Omron CX-Programmer project NewProject (CX-Programmer 9.75)

# PLC NewPLC1: CP1H XA

## Global symbols (name address type ; comment)
0 CHANNEL  ; ASSEMBLED AND DISSASSEMBLED
13.01 BOOL  ; FRGTGHN
13.05 BOOL  ; reset1
17.02 BOOL  ; reset2
265.00 BOOL  ; FEEDING BASE HMI
266.00 BOOL  ; ASSEMBLING THE BEARING
267.01 BOOL  ; INSERTION OF THE SHAFT
269.00 BOOL  ; POSITIONING OF THE COVER
278.00 BOOL  ; RUN
400.00 BOOL  ; run
C0000 BOOL  ; cup
D100 CHANNEL  ; MOV2
D105 CHANNEL  ; MOV1
D80 CHANNEL  ; .....
T0030 BOOL  ; TIMER30
W0 CHANNEL  ; ..;;,
W1 CHANNEL  ; EF

## Program NewProgram1 (cyclic task 0)
Local symbols
APLUS 100.00 BOOL  ; Feeder cylinder forwards
BPLUS 100.01 BOOL  ; Body transfer cylinder forwards
CPLUS 100.02 BOOL  ; Position verification cylinder downwards
DPLUS 100.03 BOOL  ; Rejection cylinder forwards
EMINUS 100.05 BOOL  ; Rotary actuator backwards
EPLUS 100.04 BOOL  ; Rotary actuator forwards
FM 101.06 BOOL  ; Error light on
FPLUS 100.06 BOOL  ; Opening of the gripper of the rotary actuator
GPLUS 100.07 BOOL  ; Shaft insertion manipulator downwards
HPLUS 101.00 BOOL  ; Shaft insertion manipulator forwards
IPLUS 101.01 BOOL  ; Gripper closure
JMINUS 101.03 BOOL  ; Cover insertion manipulator backwards
JPLUS 101.02 BOOL  ; Cover insertion manipulator forwards
KPLUS 101.04 BOOL  ; Cover insertion manipulator downwards
Step_0 H0.00 BOOL  ; Step 0
Step_1 H0.01 BOOL  ; Step  1
Step_10 H0.10 BOOL  ; Step 10
Step_11 H0.11 BOOL  ; Step 11
Step_12 H0.12 BOOL  ; Step 12
Step_13 H0.13 BOOL  ; Step 13
Step_14 H0.14 BOOL  ; Step 14
Step_15 H0.15 BOOL  ; Step 15
Step_16 H1.00 BOOL  ; Step 16
Step_17 H1.01 BOOL  ; Step 17
Step_18 H1.02 BOOL  ; Step 18
Step_19 H1.03 BOOL  ; Step 19
Step_2 H0.02 BOOL  ; Step 2
Step_20 H1.04 BOOL  ; Step 20
Step_21 H1.05 BOOL  ; Step 21
Step_22 H1.06 BOOL  ; Step 22
Step_23 H1.07 BOOL  ; Step 23
Step_24 H1.08 BOOL  ; Step 24
Step_25 H1.09 BOOL  ; Step 25
Step_26 H1.10 BOOL  ; Step 26
Step_27 H1.11 BOOL  ; Step 27
Step_28 H1.12 BOOL  ; Step 28
Step_29 H1.13 BOOL  ; Step 29
Step_3 H0.03 BOOL  ; Step 3
Step_30 H1.14 BOOL  ; Step 30
Step_31 H1.15 BOOL  ; Step 31
Step_32 H2.00 BOOL  ; Step 32
Step_33 H2.01 BOOL  ; Step 33
Step_34 H2.02 BOOL  ; Step 34
Step_35 H2.03 BOOL  ; Step 35
Step_36 H2.04 BOOL  ; Step 36
Step_37 H2.05 BOOL  ; Step 37
Step_38 H2.06 BOOL  ; Step 38
Step_39 H2.07 BOOL  ; Step 39
Step_4 H0.04 BOOL  ; Step 4
Step_40 H2.08 BOOL  ; Step 40
Step_41 H2.09 BOOL  ; Step 41
Step_42 H2.10 BOOL  ; Step 42
Step_43 H2.11 BOOL  ; Step 43
Step_44 H2.12 BOOL  ; Step 44
Step_45 H2.13 BOOL  ; Step 45
Step_46 H2.14 BOOL  ; Step 46
Step_47 H2.15 BOOL  ; Step 47
Step_48 H3.00 BOOL  ; Step 48
Step_49 H3.01 BOOL  ; Step 49
Step_5 H0.05 BOOL  ; Step 5
Step_50 H3.02 BOOL  ; Step 50
Step_51 H3.03 BOOL  ; Step 51
Step_6 H0.06 BOOL  ; Step 6
Step_60 H3.04 BOOL  ; Step 60
Step_61 H3.05 BOOL  ; Step 61
Step_62 H3.06 BOOL  ; Step 62
Step_7 H0.07 BOOL  ; Step 7
Step_8 H0.08 BOOL  ; Step 8
Step_9 H0.09 BOOL  ; Step 9
VPLUS 101.05 BOOL  ; Vacuum in cups
a_0 0.03 BOOL  ; Body Feeder backward
a_1 0.04 BOOL  ; Body Feeder forward
am_SCADA 20.02 BOOL  ; Auto/manu selector from SCADA
atm 0.02 BOOL  ; Auto/Manu selector
b_1 0.05 BOOL  ; Body transfer cylinder forward
bearing_placed 200.10 BOOL  ; bearing placed on body
body_ok 200.04 BOOL  ; Body placed ok
c_1 0.06 BOOL  ; Position verification cylinder downward
continue 200.01 BOOL  ; Continue cycle from one step to another
cover 200.02 BOOL  ; cover in position
cover_placed 200.09 BOOL  ; cover placed on body
cycle H4.00 BOOL  ; Cycle started
cycle_end 200.11 BOOL  ; cycle end
cycle_start 30.07 BOOL  ; cycle start
dp1 1.09 BOOL  ; Body detector
dp2 1.10 BOOL  ; Bearing detector
dp3 1.11 BOOL  ; Shaft detector
dp4 200.08 BOOL  ; Cover detector
e_0 0.07 BOOL  ; Rotary actuator backward
e_1 0.08 BOOL  ; Rotary actuator in the middle position
e_2 0.09 BOOL  ; Rotary actuator forward
error 200.12 BOOL  ; Error in the station
g_0 0.10 BOOL  ; Shaft insertion manipulator upward
g_1 0.11 BOOL  ; Shaft insertion manipulator downward
h_0 1.00 BOOL  ; Shaft insertion manipulator backward
h_1 1.01 BOOL  ; Shaft insertion manipulator forward
i_0 1.02 BOOL  ; Gripper opened
i_1 1.03 BOOL  ; Gripper closed
i_c 200.03 BOOL  ; Initial condition
j_0 1.04 BOOL  ; Cover insertion manipulator backward
j_1 1.05 BOOL  ; Cover insertion manipulator forward
k_0 1.06 BOOL  ; Cover insertion manipulator upward
k_1 1.07 BOOL  ; Cover insertion manipulator downward
m 0.00 BOOL  ; Start button
m_SCADA 20.00 BOOL  ; Start button fron Scada
no_air_pressure 200.06 BOOL  ; No air pressure
no_e1 200.07 BOOL  ; Initial condition of bearing manipulator
on 200.00 BOOL  ; Start in auto mode
p 0.01 BOOL  ; Stop button
p_SCADA 20.01 BOOL  ; Stop button from Scada
shaft_placed 200.13 BOOL  ; shaft placed on body
t_0_PV T0 CHANNEL  ; Timer 0
t_0_step T0000 BOOL  ; Timer 0
t_10_PV T10 CHANNEL  ; Timer 10
t_10_step T0010 BOOL  ; Timer 10
t_11_step T0011 BOOL  ; Timer 11
t_12_step T0012 BOOL  ; Timer 12
t_13_step T0013 BOOL  ; Timer 13
t_14_step T0014 BOOL  ; Timer 14
t_15 T0015 BOOL  ; Timer 15
t_16 T0016 BOOL  ; Timer 16
t_17 T0017 BOOL  ; Timer 17
t_18 T0018 BOOL  ; Timer 18
t_19 T0019 BOOL  ; Timer 19
t_1_PV T1 CHANNEL  ; Timer 1
t_1_step T0001 BOOL  ; Timer 1
t_20 T0020 BOOL  ; Timer 20
t_21 T0021 BOOL  ; Timer 21
t_22 T0022 BOOL  ; Timer 22
t_23 T0023 BOOL  ; Timer 23
t_24 T0024 BOOL  ; Timer 24
t_2_PV T2 CHANNEL  ; Timer 2
t_2_step T0002 BOOL  ; Timer 2
t_3_PV T3 CHANNEL  ; Timer 3
t_3_step T0003 BOOL  ; Timer 3
t_4_PV T4 CHANNEL  ; Timer 4
t_4_step T0004 BOOL  ; Timer 4
t_5_PV T5 CHANNEL  ; Timer 5
t_5_step T0005 BOOL  ; Timer 5
t_6_PV T6 CHANNEL  ; Timer 6
t_6_step T0006 BOOL  ; Timer 6
t_7 BOOL
t_7_PV T7 CHANNEL  ; Timer 7
t_7_step T0007 BOOL  ; Timer 7
t_8_PV T8 CHANNEL  ; Timer 8
t_8_step T0008 BOOL  ; Timer 8
t_9_PV T9 CHANNEL  ; Timer 9
t_9_step T0009 BOOL  ; Timer 9
v 1.08 BOOL  ; Vacuum in cups
wait 200.05 BOOL  ; Wait to return subroutine

### Section Steps

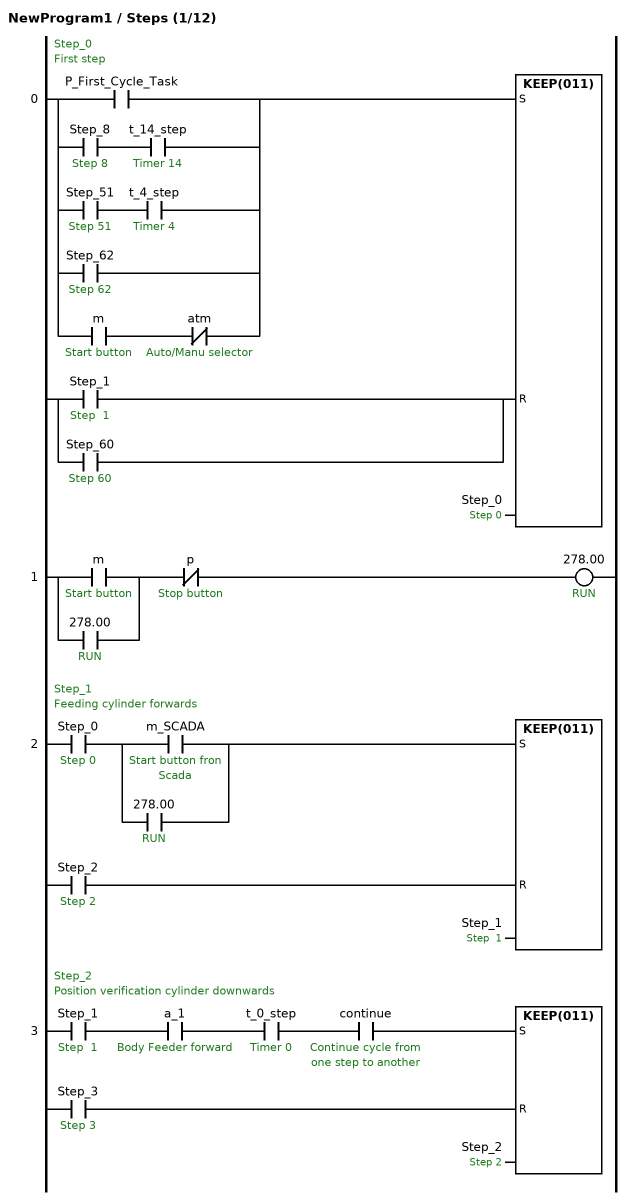
; rung 0: Step_0 / First step
LD P_First_Cycle_Task
LD Step_8  ; Step 8
AND t_14_step  ; Timer 14
ORLD
LD Step_51  ; Step 51
AND t_4_step  ; Timer 4
ORLD
OR Step_62  ; Step 62
LD m  ; Start button
ANDNOT atm  ; Auto/Manu selector
ORLD
LD Step_1  ; Step  1
OR Step_60  ; Step 60
KEEP(011) Step_0  ; Step 0
; rung 1
LD m  ; Start button
OR 278.00  ; RUN
ANDNOT p  ; Stop button
OUT 278.00  ; RUN
; rung 2: Step_1 / Feeding cylinder forwards
LD Step_0  ; Step 0
LD m_SCADA  ; Start button fron Scada
OR 278.00  ; RUN
ANDLD
LD Step_2  ; Step 2
KEEP(011) Step_1  ; Step  1
; rung 3: Step_2 / Position verification cylinder downwards
LD Step_1  ; Step  1
AND a_1  ; Body Feeder forward
AND t_0_step  ; Timer 0
AND continue  ; Continue cycle from one step to another
LD Step_3  ; Step 3
KEEP(011) Step_2  ; Step 2

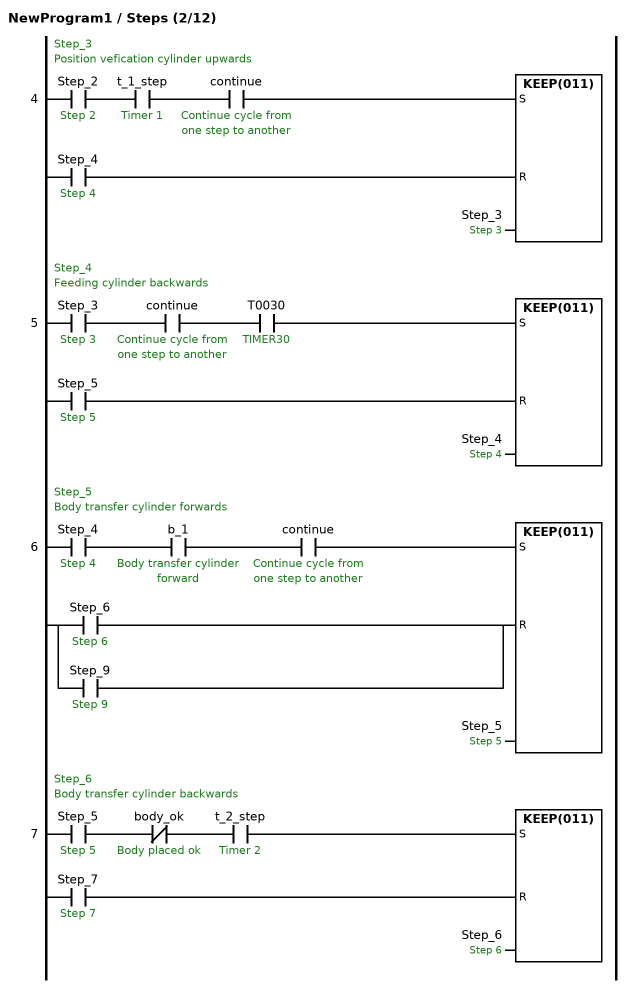
; rung 4: Step_3 / Position vefication cylinder upwards
LD Step_2  ; Step 2
AND t_1_step  ; Timer 1
AND continue  ; Continue cycle from one step to another
LD Step_4  ; Step 4
KEEP(011) Step_3  ; Step 3
; rung 5: Step_4 / Feeding cylinder backwards
LD Step_3  ; Step 3
AND continue  ; Continue cycle from one step to another
AND T0030  ; TIMER30
LD Step_5  ; Step 5
KEEP(011) Step_4  ; Step 4
; rung 6: Step_5 / Body transfer cylinder forwards
LD Step_4  ; Step 4
AND b_1  ; Body transfer cylinder forward
AND continue  ; Continue cycle from one step to another
LD Step_6  ; Step 6
OR Step_9  ; Step 9
KEEP(011) Step_5  ; Step 5
; rung 7: Step_6 / Body transfer cylinder backwards
LD Step_5  ; Step 5
ANDNOT body_ok  ; Body placed ok
AND t_2_step  ; Timer 2
LD Step_7  ; Step 7
KEEP(011) Step_6  ; Step 6

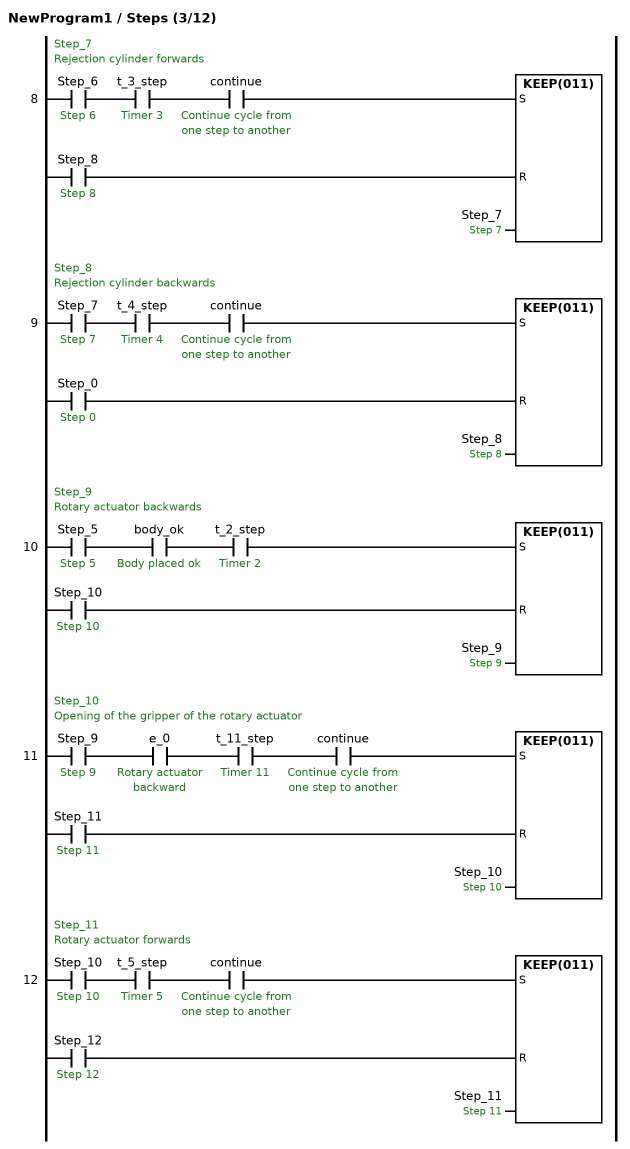
; rung 8: Step_7 / Rejection cylinder forwards
LD Step_6  ; Step 6
AND t_3_step  ; Timer 3
AND continue  ; Continue cycle from one step to another
LD Step_8  ; Step 8
KEEP(011) Step_7  ; Step 7
; rung 9: Step_8 / Rejection cylinder backwards
LD Step_7  ; Step 7
AND t_4_step  ; Timer 4
AND continue  ; Continue cycle from one step to another
LD Step_0  ; Step 0
KEEP(011) Step_8  ; Step 8
; rung 10: Step_9 / Rotary actuator backwards
LD Step_5  ; Step 5
AND body_ok  ; Body placed ok
AND t_2_step  ; Timer 2
LD Step_10  ; Step 10
KEEP(011) Step_9  ; Step 9
; rung 11: Step_10 / Opening of the gripper of the rotary actuator
LD Step_9  ; Step 9
AND e_0  ; Rotary actuator backward
AND t_11_step  ; Timer 11
AND continue  ; Continue cycle from one step to another
LD Step_11  ; Step 11
KEEP(011) Step_10  ; Step 10
; rung 12: Step_11 / Rotary actuator forwards
LD Step_10  ; Step 10
AND t_5_step  ; Timer 5
AND continue  ; Continue cycle from one step to another
LD Step_12  ; Step 12
KEEP(011) Step_11  ; Step 11

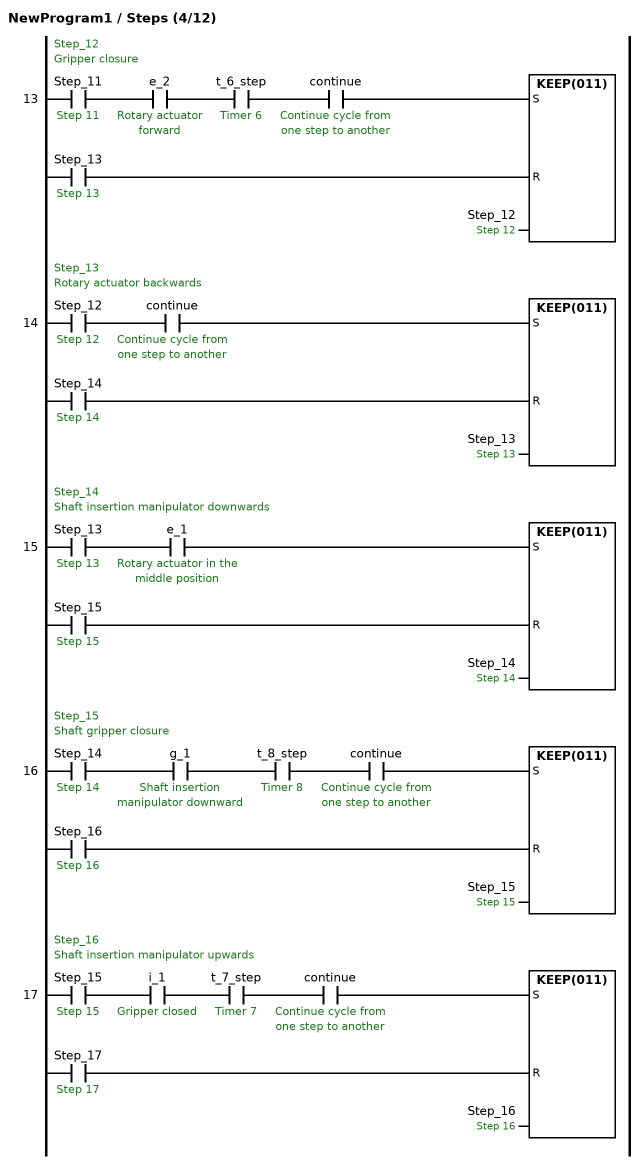
; rung 13: Step_12 / Gripper closure
LD Step_11  ; Step 11
AND e_2  ; Rotary actuator forward
AND t_6_step  ; Timer 6
AND continue  ; Continue cycle from one step to another
LD Step_13  ; Step 13
KEEP(011) Step_12  ; Step 12
; rung 14: Step_13 / Rotary actuator backwards
LD Step_12  ; Step 12
AND continue  ; Continue cycle from one step to another
LD Step_14  ; Step 14
KEEP(011) Step_13  ; Step 13
; rung 15: Step_14 / Shaft insertion manipulator downwards
LD Step_13  ; Step 13
AND e_1  ; Rotary actuator in the middle position
LD Step_15  ; Step 15
KEEP(011) Step_14  ; Step 14
; rung 16: Step_15 / Shaft gripper closure
LD Step_14  ; Step 14
AND g_1  ; Shaft insertion manipulator downward
AND t_8_step  ; Timer 8
AND continue  ; Continue cycle from one step to another
LD Step_16  ; Step 16
KEEP(011) Step_15  ; Step 15
; rung 17: Step_16 / Shaft insertion manipulator upwards
LD Step_15  ; Step 15
AND i_1  ; Gripper closed
AND t_7_step  ; Timer 7
AND continue  ; Continue cycle from one step to another
LD Step_17  ; Step 17
KEEP(011) Step_16  ; Step 16

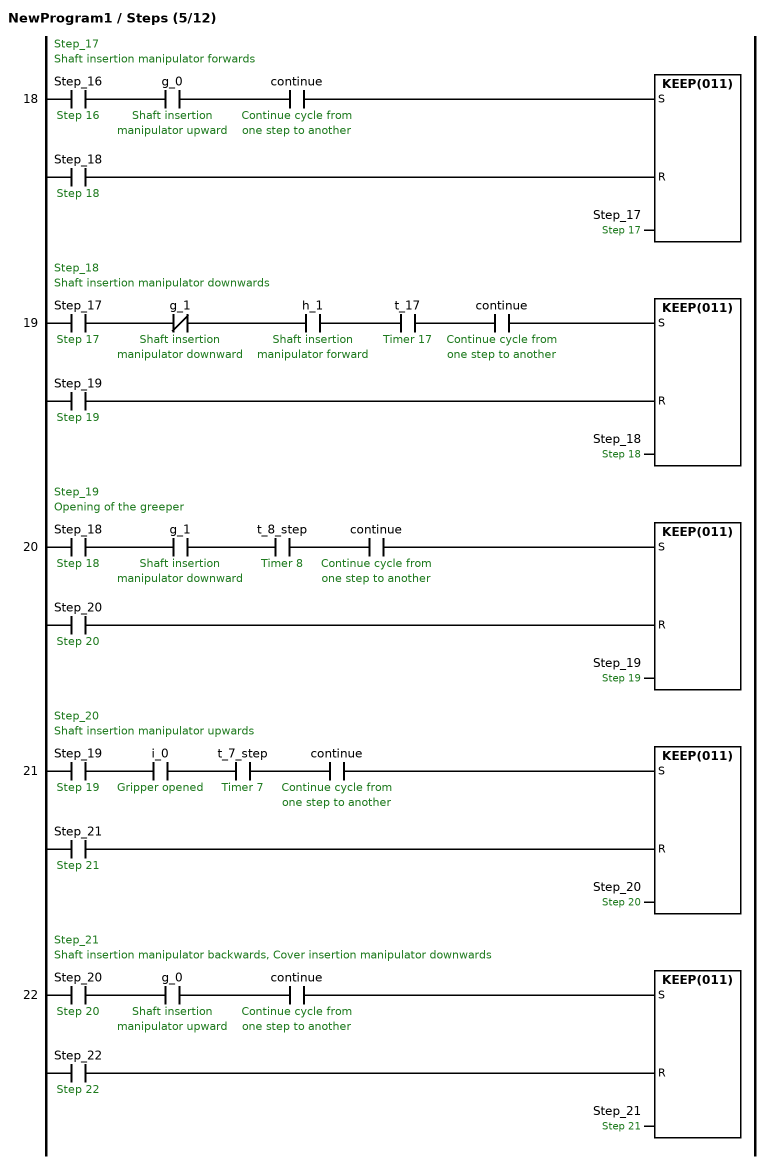
; rung 18: Step_17 / Shaft insertion manipulator forwards
LD Step_16  ; Step 16
AND g_0  ; Shaft insertion manipulator upward
AND continue  ; Continue cycle from one step to another
LD Step_18  ; Step 18
KEEP(011) Step_17  ; Step 17
; rung 19: Step_18 / Shaft insertion manipulator downwards
LD Step_17  ; Step 17
ANDNOT g_1  ; Shaft insertion manipulator downward
AND h_1  ; Shaft insertion manipulator forward
AND t_17  ; Timer 17
AND continue  ; Continue cycle from one step to another
LD Step_19  ; Step 19
KEEP(011) Step_18  ; Step 18
; rung 20: Step_19 / Opening of the greeper
LD Step_18  ; Step 18
AND g_1  ; Shaft insertion manipulator downward
AND t_8_step  ; Timer 8
AND continue  ; Continue cycle from one step to another
LD Step_20  ; Step 20
KEEP(011) Step_19  ; Step 19
; rung 21: Step_20 / Shaft insertion manipulator upwards
LD Step_19  ; Step 19
AND i_0  ; Gripper opened
AND t_7_step  ; Timer 7
AND continue  ; Continue cycle from one step to another
LD Step_21  ; Step 21
KEEP(011) Step_20  ; Step 20
; rung 22: Step_21 / Shaft insertion manipulator backwards, Cover insertion manipulator downwards
LD Step_20  ; Step 20
AND g_0  ; Shaft insertion manipulator upward
AND continue  ; Continue cycle from one step to another
LD Step_22  ; Step 22
KEEP(011) Step_21  ; Step 21

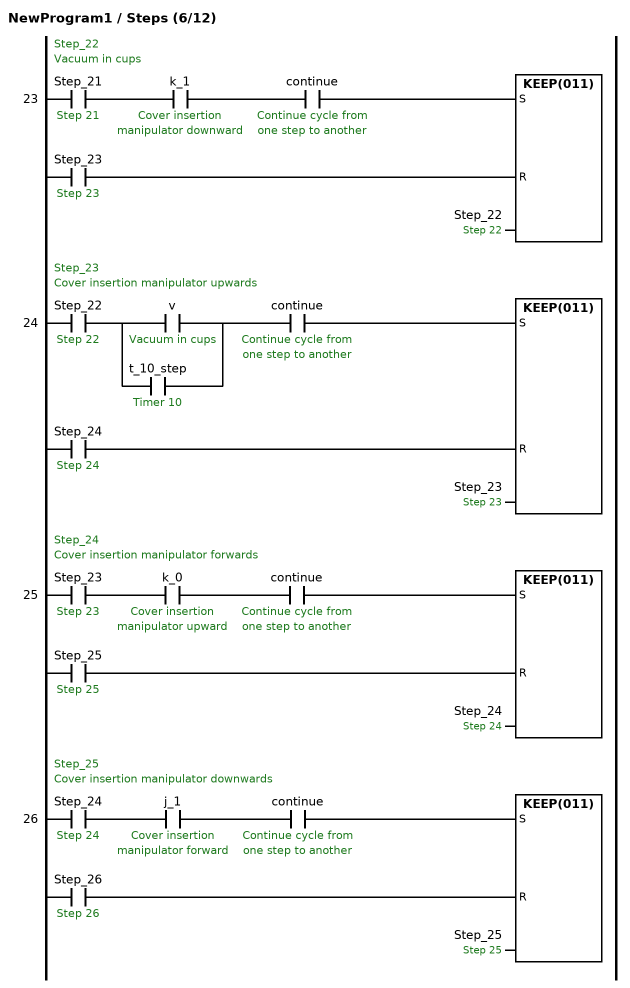
; rung 23: Step_22 / Vacuum in cups
LD Step_21  ; Step 21
AND k_1  ; Cover insertion manipulator downward
AND continue  ; Continue cycle from one step to another
LD Step_23  ; Step 23
KEEP(011) Step_22  ; Step 22
; rung 24: Step_23 / Cover insertion manipulator upwards
LD Step_22  ; Step 22
LD v  ; Vacuum in cups
OR t_10_step  ; Timer 10
ANDLD
AND continue  ; Continue cycle from one step to another
LD Step_24  ; Step 24
KEEP(011) Step_23  ; Step 23
; rung 25: Step_24 / Cover insertion manipulator forwards
LD Step_23  ; Step 23
AND k_0  ; Cover insertion manipulator upward
AND continue  ; Continue cycle from one step to another
LD Step_25  ; Step 25
KEEP(011) Step_24  ; Step 24
; rung 26: Step_25 / Cover insertion manipulator downwards
LD Step_24  ; Step 24
AND j_1  ; Cover insertion manipulator forward
AND continue  ; Continue cycle from one step to another
LD Step_26  ; Step 26
KEEP(011) Step_25  ; Step 25

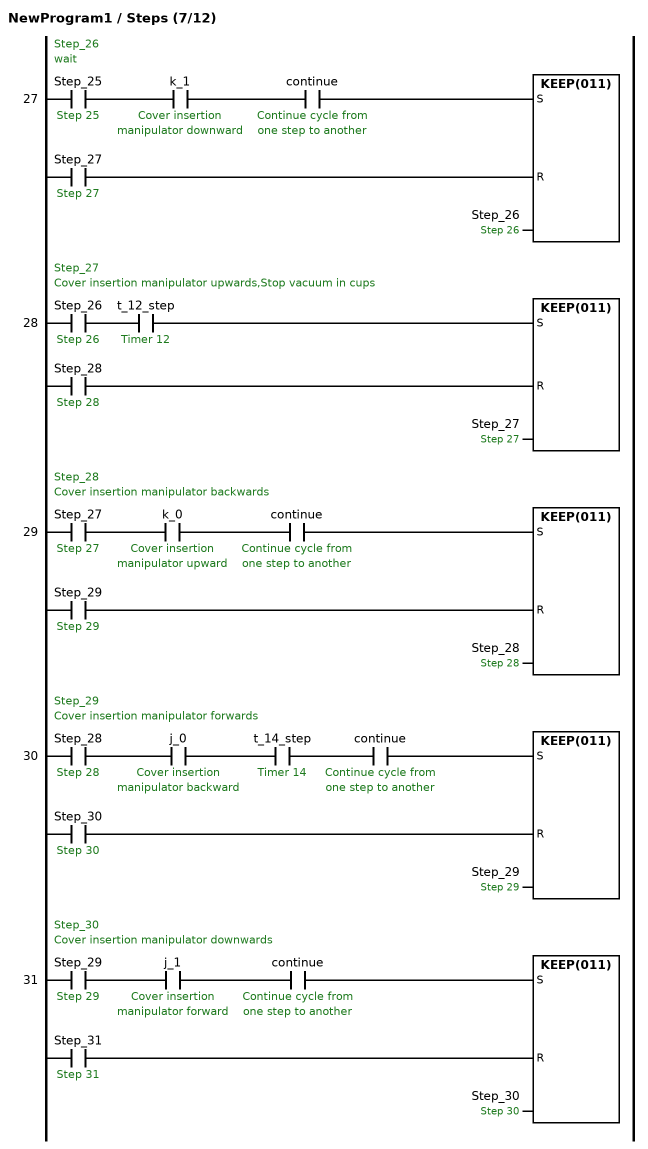
; rung 27: Step_26 / wait
LD Step_25  ; Step 25
AND k_1  ; Cover insertion manipulator downward
AND continue  ; Continue cycle from one step to another
LD Step_27  ; Step 27
KEEP(011) Step_26  ; Step 26
; rung 28: Step_27 / Cover insertion manipulator upwards,Stop vacuum in cups
LD Step_26  ; Step 26
AND t_12_step  ; Timer 12
LD Step_28  ; Step 28
KEEP(011) Step_27  ; Step 27
; rung 29: Step_28 / Cover insertion manipulator backwards
LD Step_27  ; Step 27
AND k_0  ; Cover insertion manipulator upward
AND continue  ; Continue cycle from one step to another
LD Step_29  ; Step 29
KEEP(011) Step_28  ; Step 28
; rung 30: Step_29 / Cover insertion manipulator forwards
LD Step_28  ; Step 28
AND j_0  ; Cover insertion manipulator backward
AND t_14_step  ; Timer 14
AND continue  ; Continue cycle from one step to another
LD Step_30  ; Step 30
KEEP(011) Step_29  ; Step 29
; rung 31: Step_30 / Cover insertion manipulator downwards
LD Step_29  ; Step 29
AND j_1  ; Cover insertion manipulator forward
AND continue  ; Continue cycle from one step to another
LD Step_31  ; Step 31
KEEP(011) Step_30  ; Step 30

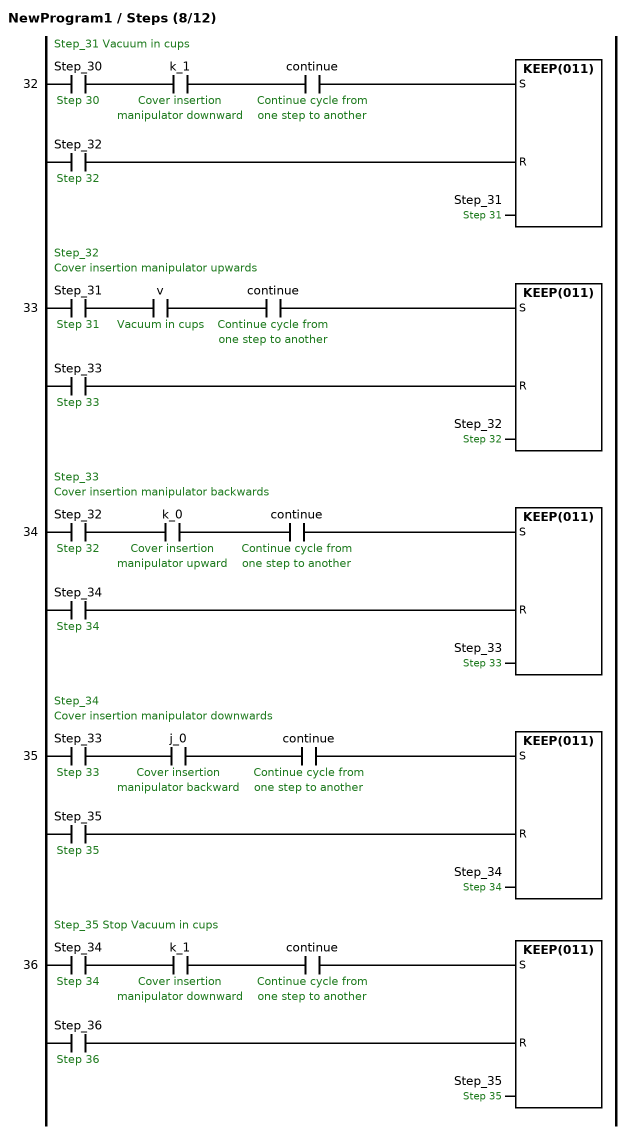
; rung 32: Step_31 Vacuum in cups
LD Step_30  ; Step 30
AND k_1  ; Cover insertion manipulator downward
AND continue  ; Continue cycle from one step to another
LD Step_32  ; Step 32
KEEP(011) Step_31  ; Step 31
; rung 33: Step_32 / Cover insertion manipulator upwards
LD Step_31  ; Step 31
AND v  ; Vacuum in cups
AND continue  ; Continue cycle from one step to another
LD Step_33  ; Step 33
KEEP(011) Step_32  ; Step 32
; rung 34: Step_33 / Cover insertion manipulator backwards
LD Step_32  ; Step 32
AND k_0  ; Cover insertion manipulator upward
AND continue  ; Continue cycle from one step to another
LD Step_34  ; Step 34
KEEP(011) Step_33  ; Step 33
; rung 35: Step_34 / Cover insertion manipulator downwards
LD Step_33  ; Step 33
AND j_0  ; Cover insertion manipulator backward
AND continue  ; Continue cycle from one step to another
LD Step_35  ; Step 35
KEEP(011) Step_34  ; Step 34
; rung 36: Step_35 Stop Vacuum in cups
LD Step_34  ; Step 34
AND k_1  ; Cover insertion manipulator downward
AND continue  ; Continue cycle from one step to another
LD Step_36  ; Step 36
KEEP(011) Step_35  ; Step 35

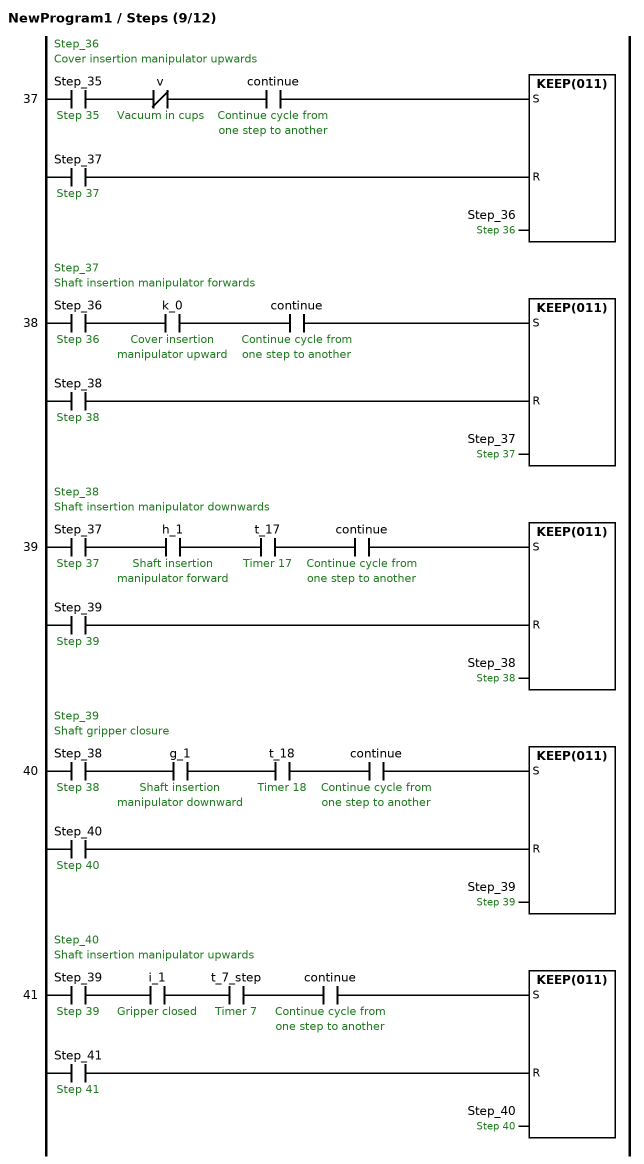
; rung 37: Step_36 / Cover insertion manipulator upwards
LD Step_35  ; Step 35
ANDNOT v  ; Vacuum in cups
AND continue  ; Continue cycle from one step to another
LD Step_37  ; Step 37
KEEP(011) Step_36  ; Step 36
; rung 38: Step_37 / Shaft insertion manipulator forwards
LD Step_36  ; Step 36
AND k_0  ; Cover insertion manipulator upward
AND continue  ; Continue cycle from one step to another
LD Step_38  ; Step 38
KEEP(011) Step_37  ; Step 37
; rung 39: Step_38 / Shaft insertion manipulator downwards
LD Step_37  ; Step 37
AND h_1  ; Shaft insertion manipulator forward
AND t_17  ; Timer 17
AND continue  ; Continue cycle from one step to another
LD Step_39  ; Step 39
KEEP(011) Step_38  ; Step 38
; rung 40: Step_39 / Shaft gripper closure
LD Step_38  ; Step 38
AND g_1  ; Shaft insertion manipulator downward
AND t_18  ; Timer 18
AND continue  ; Continue cycle from one step to another
LD Step_40  ; Step 40
KEEP(011) Step_39  ; Step 39
; rung 41: Step_40 / Shaft insertion manipulator upwards
LD Step_39  ; Step 39
AND i_1  ; Gripper closed
AND t_7_step  ; Timer 7
AND continue  ; Continue cycle from one step to another
LD Step_41  ; Step 41
KEEP(011) Step_40  ; Step 40

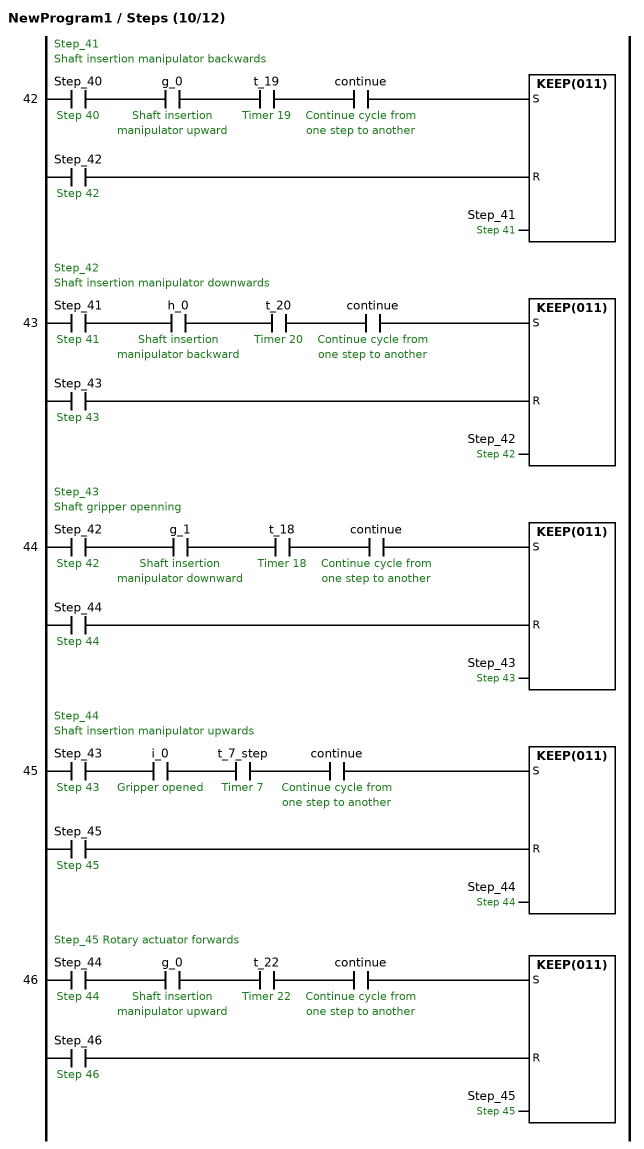
; rung 42: Step_41 / Shaft insertion manipulator backwards
LD Step_40  ; Step 40
AND g_0  ; Shaft insertion manipulator upward
AND t_19  ; Timer 19
AND continue  ; Continue cycle from one step to another
LD Step_42  ; Step 42
KEEP(011) Step_41  ; Step 41
; rung 43: Step_42 / Shaft insertion manipulator downwards
LD Step_41  ; Step 41
AND h_0  ; Shaft insertion manipulator backward
AND t_20  ; Timer 20
AND continue  ; Continue cycle from one step to another
LD Step_43  ; Step 43
KEEP(011) Step_42  ; Step 42
; rung 44: Step_43 / Shaft gripper openning
LD Step_42  ; Step 42
AND g_1  ; Shaft insertion manipulator downward
AND t_18  ; Timer 18
AND continue  ; Continue cycle from one step to another
LD Step_44  ; Step 44
KEEP(011) Step_43  ; Step 43
; rung 45: Step_44 / Shaft insertion manipulator upwards
LD Step_43  ; Step 43
AND i_0  ; Gripper opened
AND t_7_step  ; Timer 7
AND continue  ; Continue cycle from one step to another
LD Step_45  ; Step 45
KEEP(011) Step_44  ; Step 44
; rung 46: Step_45 Rotary actuator forwards
LD Step_44  ; Step 44
AND g_0  ; Shaft insertion manipulator upward
AND t_22  ; Timer 22
AND continue  ; Continue cycle from one step to another
LD Step_46  ; Step 46
KEEP(011) Step_45  ; Step 45

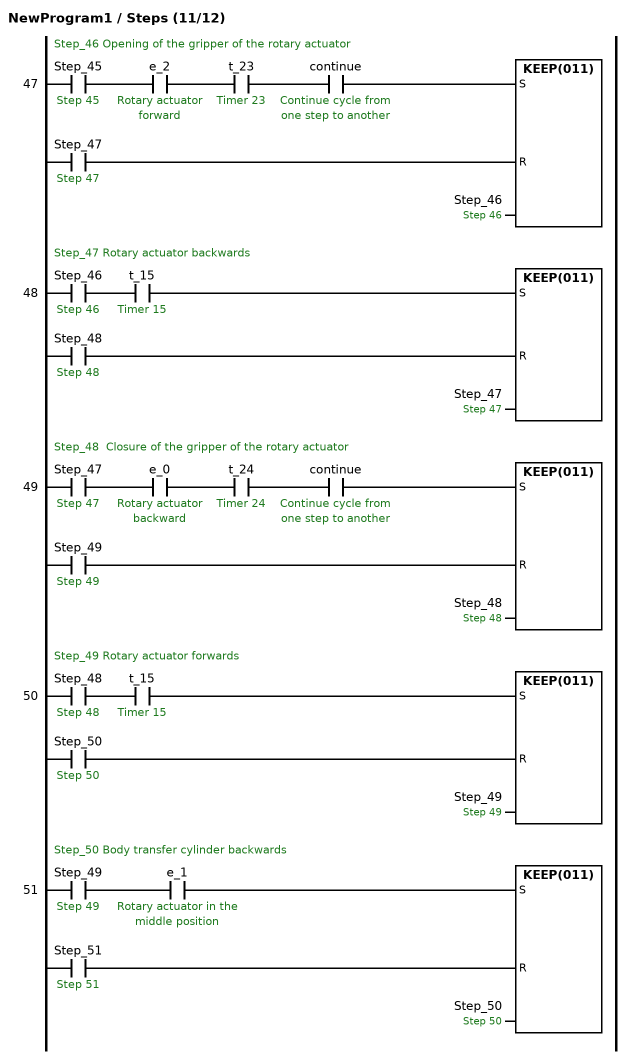
; rung 47: Step_46 Opening of the gripper of the rotary actuator
LD Step_45  ; Step 45
AND e_2  ; Rotary actuator forward
AND t_23  ; Timer 23
AND continue  ; Continue cycle from one step to another
LD Step_47  ; Step 47
KEEP(011) Step_46  ; Step 46
; rung 48: Step_47 Rotary actuator backwards
LD Step_46  ; Step 46
AND t_15  ; Timer 15
LD Step_48  ; Step 48
KEEP(011) Step_47  ; Step 47
; rung 49: Step_48  Closure of the gripper of the rotary actuator
LD Step_47  ; Step 47
AND e_0  ; Rotary actuator backward
AND t_24  ; Timer 24
AND continue  ; Continue cycle from one step to another
LD Step_49  ; Step 49
KEEP(011) Step_48  ; Step 48
; rung 50: Step_49 Rotary actuator forwards
LD Step_48  ; Step 48
AND t_15  ; Timer 15
LD Step_50  ; Step 50
KEEP(011) Step_49  ; Step 49
; rung 51: Step_50 Body transfer cylinder backwards
LD Step_49  ; Step 49
AND e_1  ; Rotary actuator in the middle position
LD Step_51  ; Step 51
KEEP(011) Step_50  ; Step 50

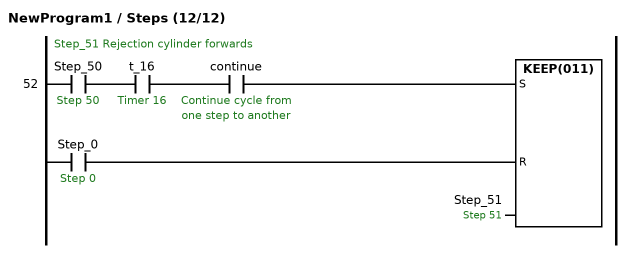
; rung 52: Step_51 Rejection cylinder forwards
LD Step_50  ; Step 50
AND t_16  ; Timer 16
AND continue  ; Continue cycle from one step to another
LD Step_0  ; Step 0
KEEP(011) Step_51  ; Step 51

### Section Outputs

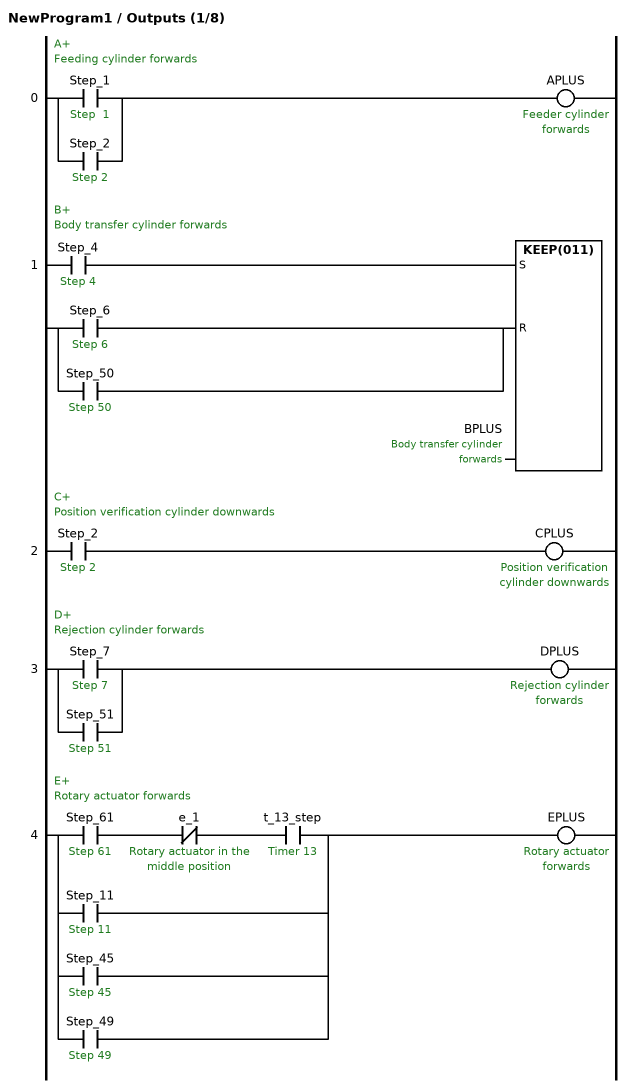
; rung 0: A+ / Feeding cylinder forwards
LD Step_1  ; Step  1
OR Step_2  ; Step 2
OUT APLUS  ; Feeder cylinder forwards
; rung 1: B+ / Body transfer cylinder forwards
LD Step_4  ; Step 4
LD Step_6  ; Step 6
OR Step_50  ; Step 50
KEEP(011) BPLUS  ; Body transfer cylinder forwards
; rung 2: C+ / Position verification cylinder downwards
LD Step_2  ; Step 2
OUT CPLUS  ; Position verification cylinder downwards
; rung 3: D+ / Rejection cylinder forwards
LD Step_7  ; Step 7
OR Step_51  ; Step 51
OUT DPLUS  ; Rejection cylinder forwards
; rung 4: E+ / Rotary actuator forwards
LD Step_61  ; Step 61
ANDNOT e_1  ; Rotary actuator in the middle position
AND t_13_step  ; Timer 13
OR Step_11  ; Step 11
OR Step_45  ; Step 45
OR Step_49  ; Step 49
OUT EPLUS  ; Rotary actuator forwards

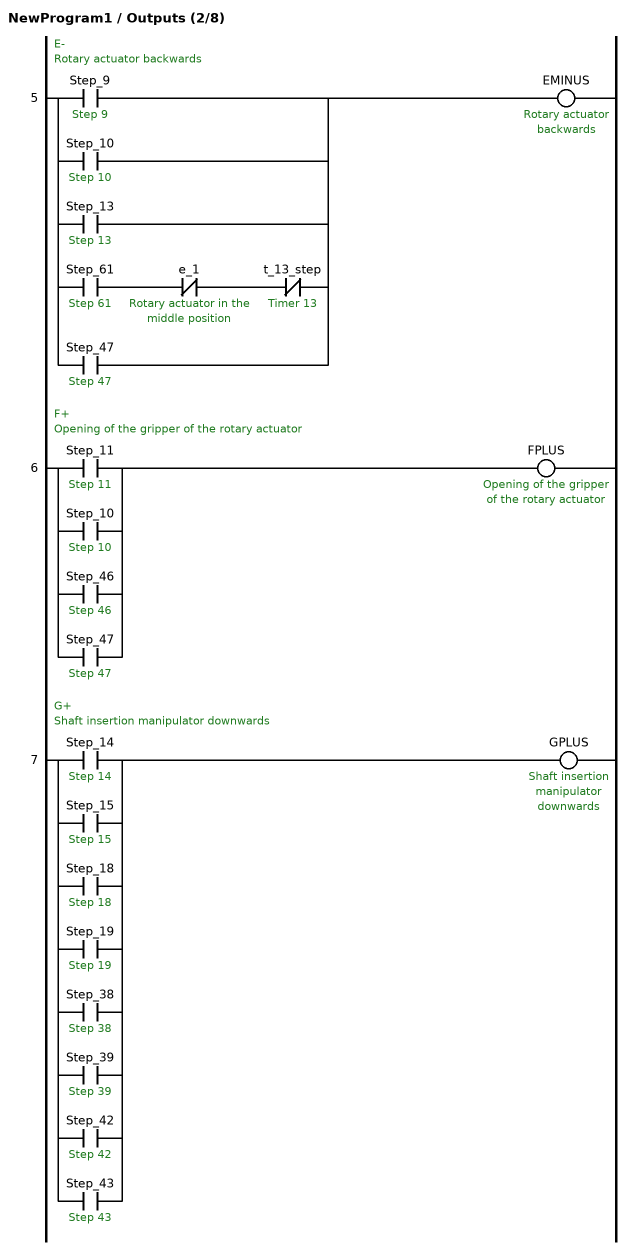
; rung 5: E- / Rotary actuator backwards
LD Step_9  ; Step 9
OR Step_10  ; Step 10
OR Step_13  ; Step 13
LD Step_61  ; Step 61
ANDNOT e_1  ; Rotary actuator in the middle position
ANDNOT t_13_step  ; Timer 13
ORLD
OR Step_47  ; Step 47
OUT EMINUS  ; Rotary actuator backwards
; rung 6: F+ / Opening of the gripper of the rotary actuator
LD Step_11  ; Step 11
OR Step_10  ; Step 10
OR Step_46  ; Step 46
OR Step_47  ; Step 47
OUT FPLUS  ; Opening of the gripper of the rotary actuator
; rung 7: G+ / Shaft insertion manipulator downwards
LD Step_14  ; Step 14
OR Step_15  ; Step 15
OR Step_18  ; Step 18
OR Step_19  ; Step 19
OR Step_38  ; Step 38
OR Step_39  ; Step 39
OR Step_42  ; Step 42
OR Step_43  ; Step 43
OUT GPLUS  ; Shaft insertion manipulator downwards

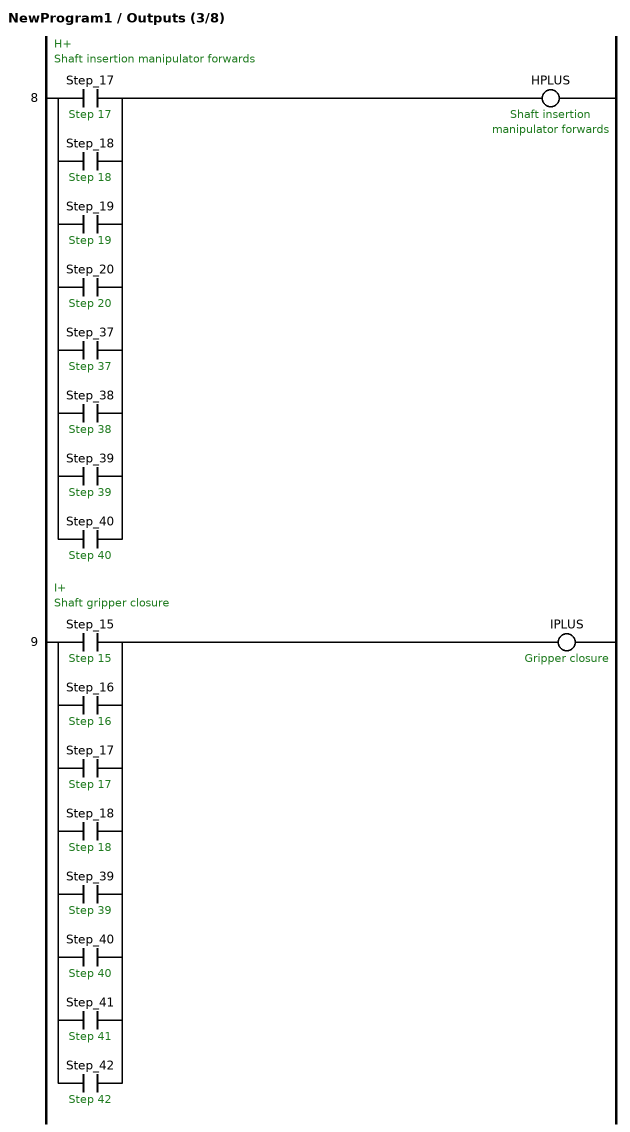
; rung 8: H+ / Shaft insertion manipulator forwards
LD Step_17  ; Step 17
OR Step_18  ; Step 18
OR Step_19  ; Step 19
OR Step_20  ; Step 20
OR Step_37  ; Step 37
OR Step_38  ; Step 38
OR Step_39  ; Step 39
OR Step_40  ; Step 40
OUT HPLUS  ; Shaft insertion manipulator forwards
; rung 9: I+ / Shaft gripper closure
LD Step_15  ; Step 15
OR Step_16  ; Step 16
OR Step_17  ; Step 17
OR Step_18  ; Step 18
OR Step_39  ; Step 39
OR Step_40  ; Step 40
OR Step_41  ; Step 41
OR Step_42  ; Step 42
OUT IPLUS  ; Gripper closure

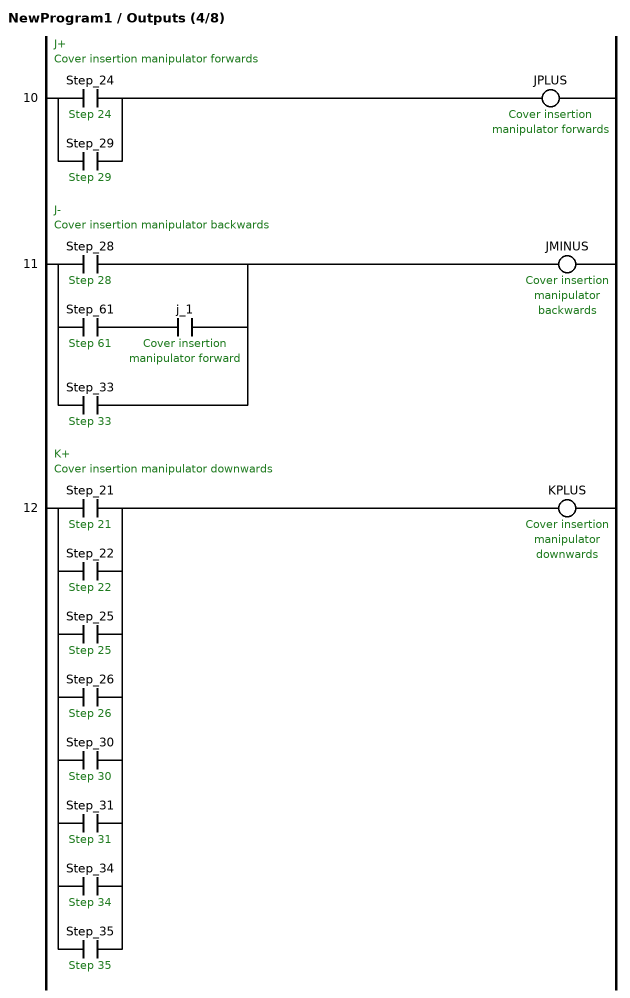
; rung 10: J+ / Cover insertion manipulator forwards
LD Step_24  ; Step 24
OR Step_29  ; Step 29
OUT JPLUS  ; Cover insertion manipulator forwards
; rung 11: J- / Cover insertion manipulator backwards
LD Step_28  ; Step 28
LD Step_61  ; Step 61
AND j_1  ; Cover insertion manipulator forward
ORLD
OR Step_33  ; Step 33
OUT JMINUS  ; Cover insertion manipulator backwards
; rung 12: K+ / Cover insertion manipulator downwards
LD Step_21  ; Step 21
OR Step_22  ; Step 22
OR Step_25  ; Step 25
OR Step_26  ; Step 26
OR Step_30  ; Step 30
OR Step_31  ; Step 31
OR Step_34  ; Step 34
OR Step_35  ; Step 35
OUT KPLUS  ; Cover insertion manipulator downwards

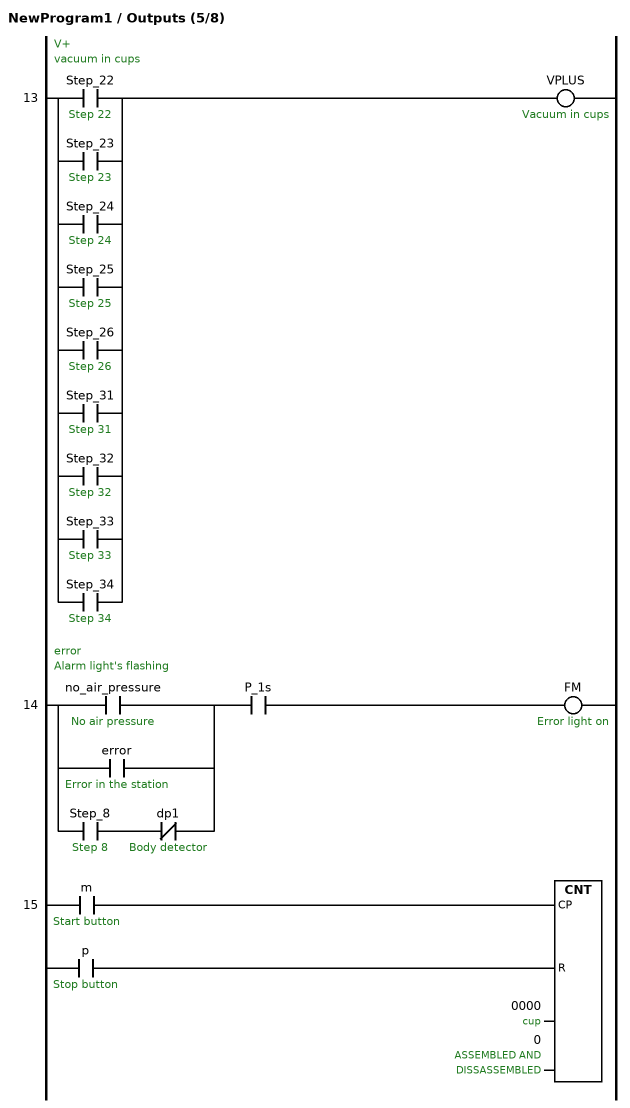
; rung 13: V+ / vacuum in cups
LD Step_22  ; Step 22
OR Step_23  ; Step 23
OR Step_24  ; Step 24
OR Step_25  ; Step 25
OR Step_26  ; Step 26
OR Step_31  ; Step 31
OR Step_32  ; Step 32
OR Step_33  ; Step 33
OR Step_34  ; Step 34
OUT VPLUS  ; Vacuum in cups
; rung 14: error / Alarm light's flashing
LD no_air_pressure  ; No air pressure
OR error  ; Error in the station
LD Step_8  ; Step 8
ANDNOT dp1  ; Body detector
ORLD
AND P_1s
OUT FM  ; Error light on
; rung 15
LD m  ; Start button
LD p  ; Stop button
CNT 0000 0  ; ASSEMBLED AND DISSASSEMBLED, cup

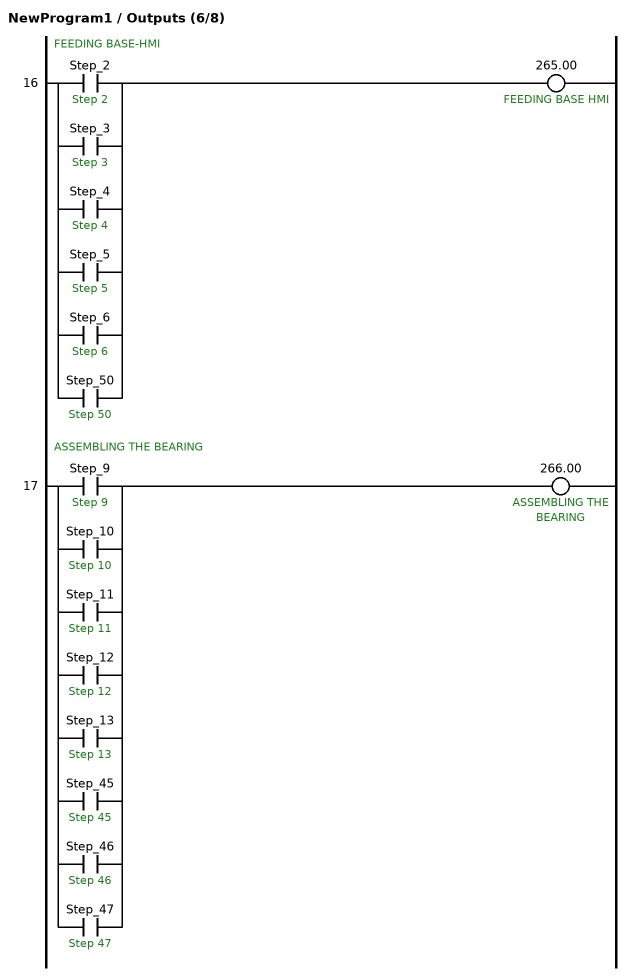
; rung 16: FEEDING BASE-HMI
LD Step_2  ; Step 2
OR Step_3  ; Step 3
OR Step_4  ; Step 4
OR Step_5  ; Step 5
OR Step_6  ; Step 6
OR Step_50  ; Step 50
OUT 265.00  ; FEEDING BASE HMI
; rung 17: ASSEMBLING THE BEARING
LD Step_9  ; Step 9
OR Step_10  ; Step 10
OR Step_11  ; Step 11
OR Step_12  ; Step 12
OR Step_13  ; Step 13
OR Step_45  ; Step 45
OR Step_46  ; Step 46
OR Step_47  ; Step 47
OUT 266.00  ; ASSEMBLING THE BEARING

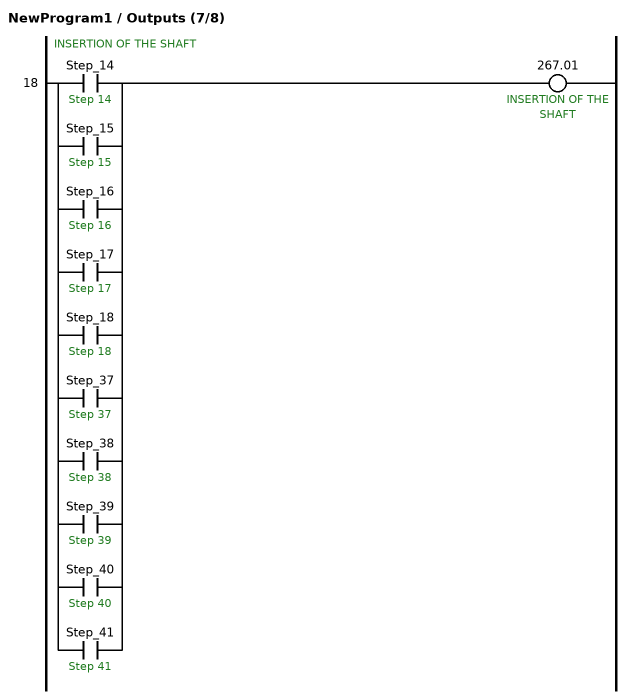
; rung 18: INSERTION OF THE SHAFT
LD Step_14  ; Step 14
OR Step_15  ; Step 15
OR Step_16  ; Step 16
OR Step_17  ; Step 17
OR Step_18  ; Step 18
OR Step_37  ; Step 37
OR Step_38  ; Step 38
OR Step_39  ; Step 39
OR Step_40  ; Step 40
OR Step_41  ; Step 41
OUT 267.01  ; INSERTION OF THE SHAFT

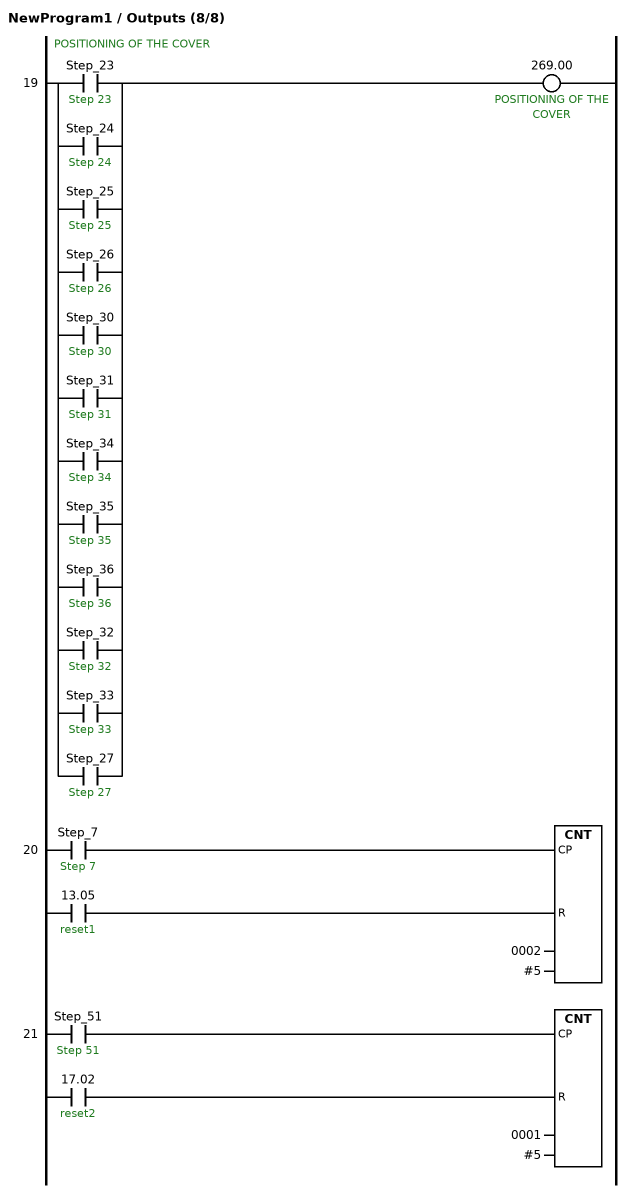
; rung 19: POSITIONING OF THE COVER
LD Step_23  ; Step 23
OR Step_24  ; Step 24
OR Step_25  ; Step 25
OR Step_26  ; Step 26
OR Step_30  ; Step 30
OR Step_31  ; Step 31
OR Step_34  ; Step 34
OR Step_35  ; Step 35
OR Step_36  ; Step 36
OR Step_32  ; Step 32
OR Step_33  ; Step 33
OR Step_27  ; Step 27
OUT 269.00  ; POSITIONING OF THE COVER
; rung 20
LD Step_7  ; Step 7
LD 13.05  ; reset1
CNT 0002 #5
; rung 21
LD Step_51  ; Step 51
LD 17.02  ; reset2
CNT 0001 #5

### Section Works_bits

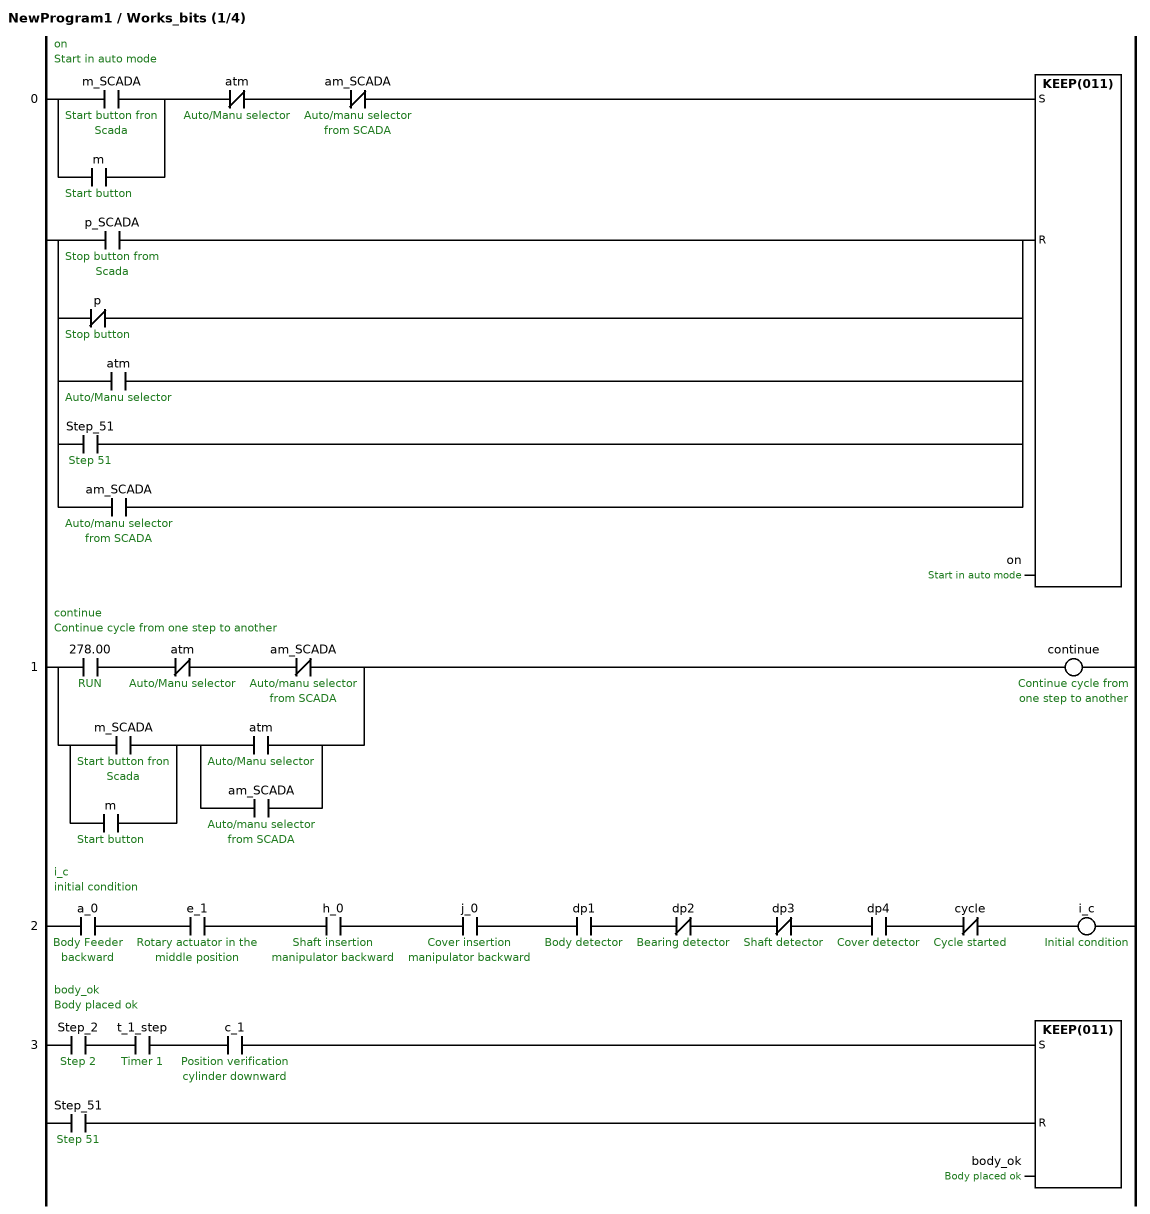
; rung 0: on / Start in auto mode
LD m_SCADA  ; Start button fron Scada
OR m  ; Start button
ANDNOT atm  ; Auto/Manu selector
ANDNOT am_SCADA  ; Auto/manu selector from SCADA
LD p_SCADA  ; Stop button from Scada
ORNOT p  ; Stop button
OR atm  ; Auto/Manu selector
OR Step_51  ; Step 51
OR am_SCADA  ; Auto/manu selector from SCADA
KEEP(011) on  ; Start in auto mode
; rung 1: continue / Continue cycle from one step to another
LD 278.00  ; RUN
ANDNOT atm  ; Auto/Manu selector
ANDNOT am_SCADA  ; Auto/manu selector from SCADA
LD m_SCADA  ; Start button fron Scada
OR m  ; Start button
LD atm  ; Auto/Manu selector
OR am_SCADA  ; Auto/manu selector from SCADA
ANDLD
ORLD
OUT continue  ; Continue cycle from one step to another
; rung 2: i_c / initial condition
LD a_0  ; Body Feeder backward
AND e_1  ; Rotary actuator in the middle position
AND h_0  ; Shaft insertion manipulator backward
AND j_0  ; Cover insertion manipulator backward
AND dp1  ; Body detector
ANDNOT dp2  ; Bearing detector
ANDNOT dp3  ; Shaft detector
AND dp4  ; Cover detector
ANDNOT cycle  ; Cycle started
OUT i_c  ; Initial condition
; rung 3: body_ok / Body placed ok
LD Step_2  ; Step 2
AND t_1_step  ; Timer 1
AND c_1  ; Position verification cylinder downward
LD Step_51  ; Step 51
KEEP(011) body_ok  ; Body placed ok

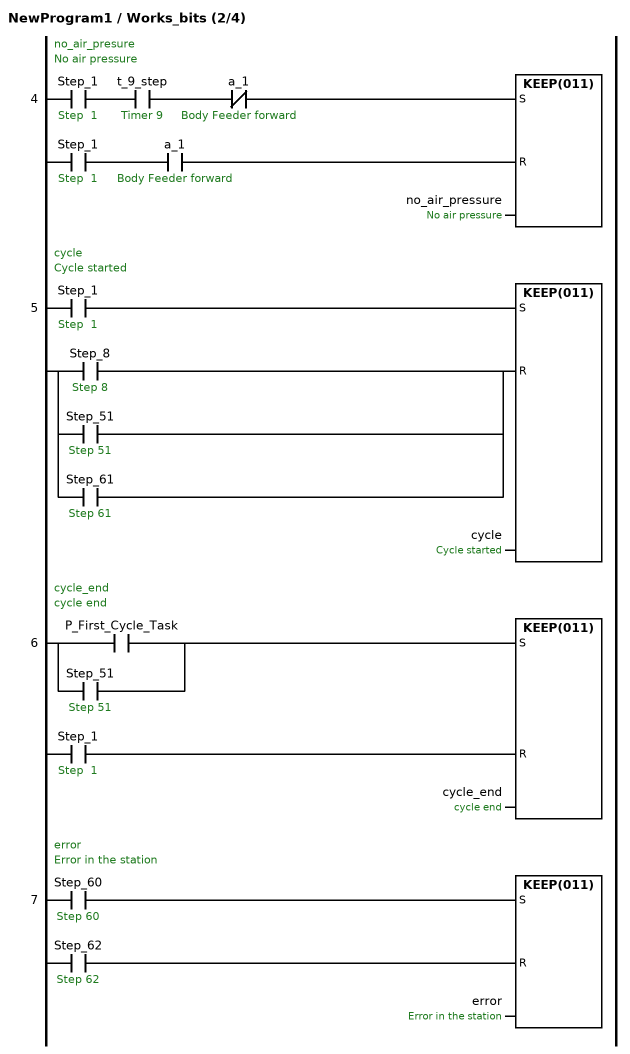
; rung 4: no_air_presure / No air pressure
LD Step_1  ; Step  1
AND t_9_step  ; Timer 9
ANDNOT a_1  ; Body Feeder forward
LD Step_1  ; Step  1
AND a_1  ; Body Feeder forward
KEEP(011) no_air_pressure  ; No air pressure
; rung 5: cycle / Cycle started
LD Step_1  ; Step  1
LD Step_8  ; Step 8
OR Step_51  ; Step 51
OR Step_61  ; Step 61
KEEP(011) cycle  ; Cycle started
; rung 6: cycle_end / cycle end
LD P_First_Cycle_Task
OR Step_51  ; Step 51
LD Step_1  ; Step  1
KEEP(011) cycle_end  ; cycle end
; rung 7: error / Error in the station
LD Step_60  ; Step 60
LD Step_62  ; Step 62
KEEP(011) error  ; Error in the station

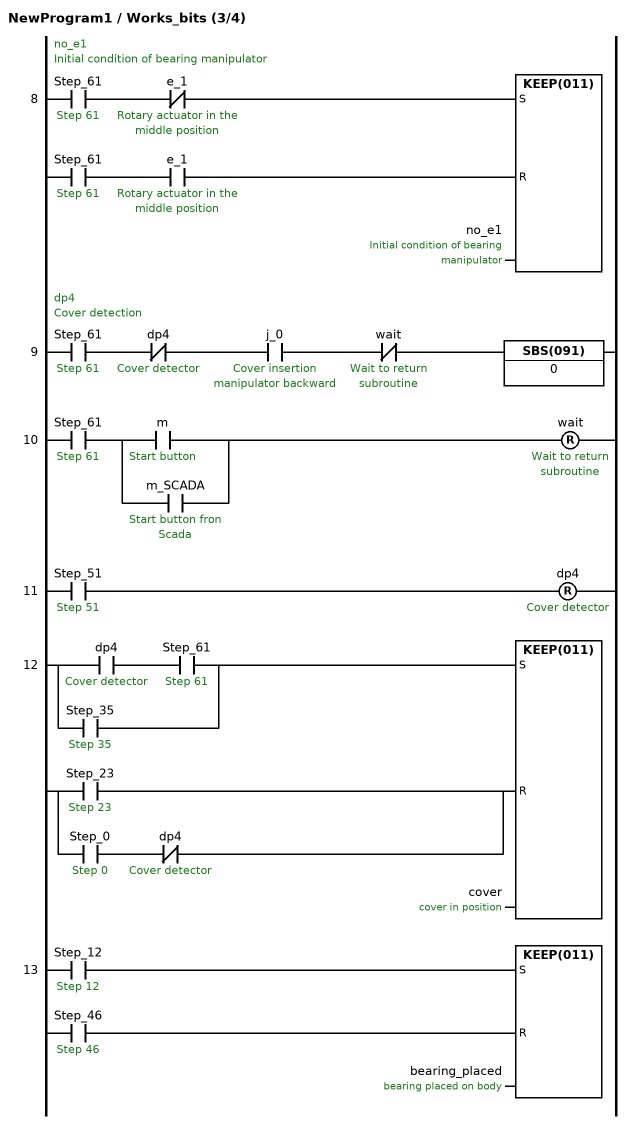
; rung 8: no_e1 / Initial condition of bearing manipulator
LD Step_61  ; Step 61
ANDNOT e_1  ; Rotary actuator in the middle position
LD Step_61  ; Step 61
AND e_1  ; Rotary actuator in the middle position
KEEP(011) no_e1  ; Initial condition of bearing manipulator
; rung 9: dp4 / Cover detection
LD Step_61  ; Step 61
ANDNOT dp4  ; Cover detector
AND j_0  ; Cover insertion manipulator backward
ANDNOT wait  ; Wait to return subroutine
SBS(091) 0
; rung 10
LD Step_61  ; Step 61
LD m  ; Start button
OR m_SCADA  ; Start button fron Scada
ANDLD
RSET wait  ; Wait to return subroutine
; rung 11
LD Step_51  ; Step 51
RSET dp4  ; Cover detector
; rung 12
LD dp4  ; Cover detector
AND Step_61  ; Step 61
OR Step_35  ; Step 35
LD Step_23  ; Step 23
LD Step_0  ; Step 0
ANDNOT dp4  ; Cover detector
ORLD
KEEP(011) cover  ; cover in position
; rung 13
LD Step_12  ; Step 12
LD Step_46  ; Step 46
KEEP(011) bearing_placed  ; bearing placed on body

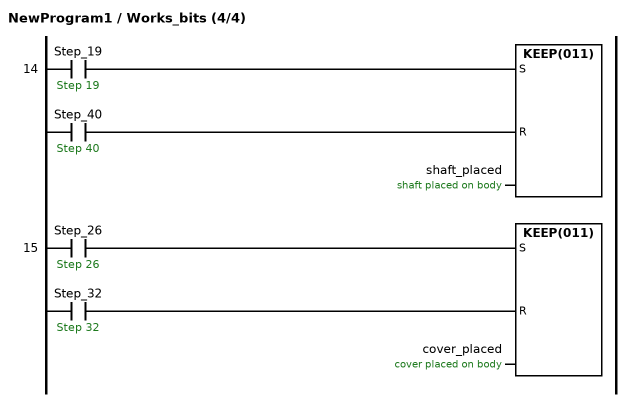
; rung 14
LD Step_19  ; Step 19
LD Step_40  ; Step 40
KEEP(011) shaft_placed  ; shaft placed on body
; rung 15
LD Step_26  ; Step 26
LD Step_32  ; Step 32
KEEP(011) cover_placed  ; cover placed on body

### Section Timers

